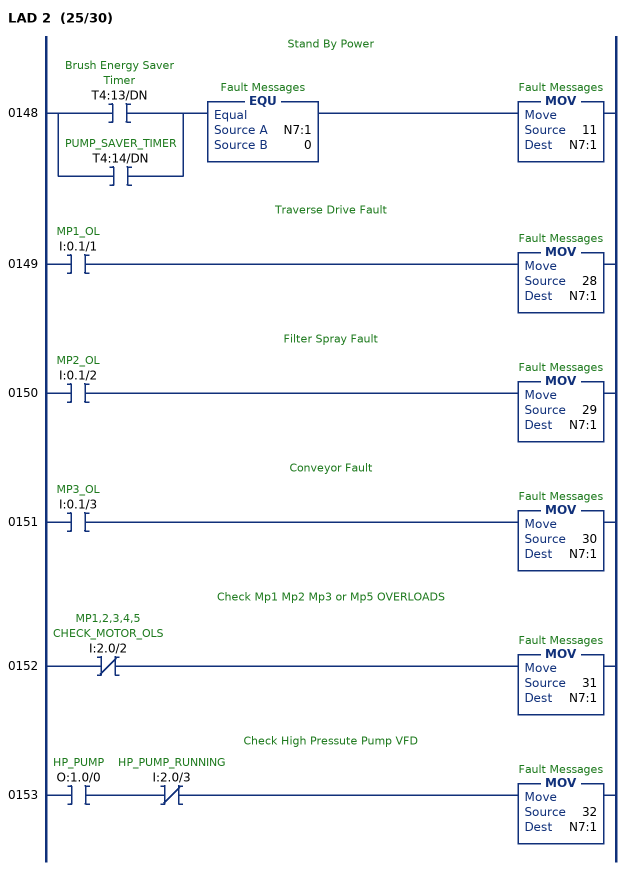
% Rung: 148 %
% Stand By Power %
SOR BST XIC T4:13/DN NXB XIC T4:14/DN BND EQU N7:1 0 MOV 11 N7:1 EOR
%   T4:13  "Brush Energy Saver Timer" %
%   T4:14/DN  PUMP_SAVER_TIMER %
%   N7:1  "Fault Messages" %
% Rung: 149 %
% Traverse Drive Fault %
SOR XIC I:0.1/1 MOV 28 N7:1 EOR
%   I:0.1/1  MP1_OL %
%   N7:1  "Fault Messages" %
% Rung: 150 %
% Filter Spray Fault %
SOR XIC I:0.1/2 MOV 29 N7:1 EOR
%   I:0.1/2  MP2_OL %
%   N7:1  "Fault Messages" %
% Rung: 151 %
% Conveyor Fault %
SOR XIC I:0.1/3 MOV 30 N7:1 EOR
%   I:0.1/3  MP3_OL %
%   N7:1  "Fault Messages" %
% Rung: 152 %
% Check Mp1 Mp2 Mp3 or Mp5 OVERLOADS %
SOR XIO I:2.0/2 MOV 31 N7:1 EOR
%   I:2.0/2  CHECK_MOTOR_OLS  "MP1,2,3,4,5" %
%   N7:1  "Fault Messages" %
% Rung: 153 %
% Check High Pressute Pump VFD %
SOR XIC O:1.0/0 XIO I:2.0/3 MOV 32 N7:1 EOR
%   O:1.0/0  HP_PUMP %
%   I:2.0/3  HP_PUMP_RUNNING %
%   N7:1  "Fault Messages" %

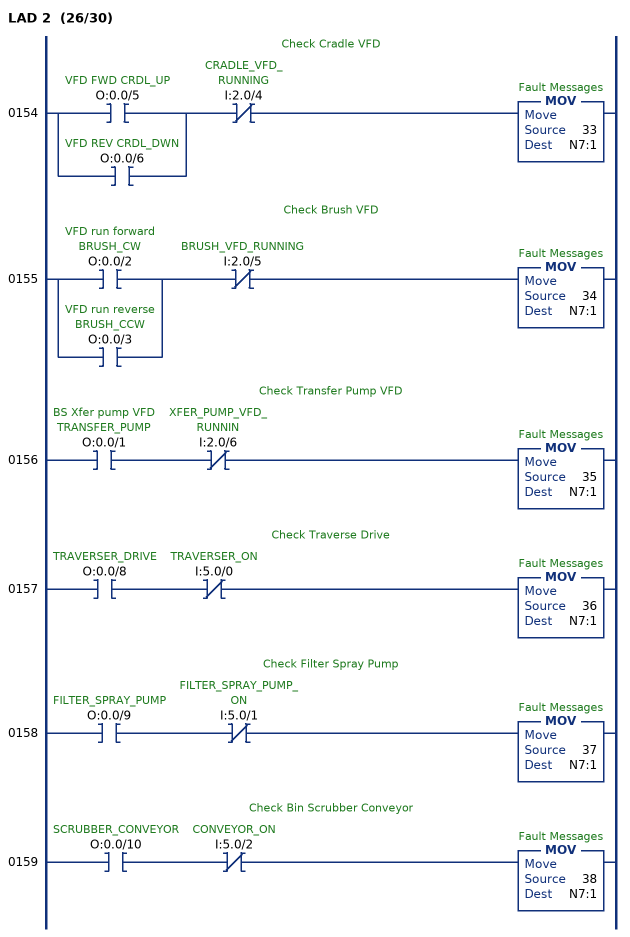
% Rung: 154 %
% Check Cradle VFD %
SOR BST XIC O:0.0/5 NXB XIC O:0.0/6 BND XIO I:2.0/4 MOV 33 N7:1 EOR
%   O:0.0/5  CRDL_UP  "VFD FWD" %
%   O:0.0/6  CRDL_DWN  "VFD REV" %
%   I:2.0/4  CRADLE_VFD_RUNNING %
%   N7:1  "Fault Messages" %
% Rung: 155 %
% Check Brush VFD %
SOR BST XIC O:0.0/2 NXB XIC O:0.0/3 BND XIO I:2.0/5 MOV 34 N7:1 EOR
%   O:0.0/2  BRUSH_CW  "VFD run forward" %
%   O:0.0/3  BRUSH_CCW  "VFD run reverse" %
%   I:2.0/5  BRUSH_VFD_RUNNING %
%   N7:1  "Fault Messages" %
% Rung: 156 %
% Check Transfer Pump VFD %
SOR XIC O:0.0/1 XIO I:2.0/6 MOV 35 N7:1 EOR
%   O:0.0/1  TRANSFER_PUMP  "BS Xfer pump VFD" %
%   I:2.0/6  XFER_PUMP_VFD_RUNNIN %
%   N7:1  "Fault Messages" %
% Rung: 157 %
% Check Traverse Drive %
SOR XIC O:0.0/8 XIO I:5.0/0 MOV 36 N7:1 EOR
%   O:0.0/8  TRAVERSER_DRIVE %
%   I:5.0/0  TRAVERSER_ON %
%   N7:1  "Fault Messages" %
% Rung: 158 %
% Check Filter Spray Pump %
SOR XIC O:0.0/9 XIO I:5.0/1 MOV 37 N7:1 EOR
%   O:0.0/9  FILTER_SPRAY_PUMP %
%   I:5.0/1  FILTER_SPRAY_PUMP_ON %
%   N7:1  "Fault Messages" %
% Rung: 159 %
% Check Bin Scrubber Conveyor %
SOR XIC O:0.0/10 XIO I:5.0/2 MOV 38 N7:1 EOR
%   O:0.0/10  SCRUBBER_CONVEYOR %
%   I:5.0/2  CONVEYOR_ON %
%   N7:1  "Fault Messages" %

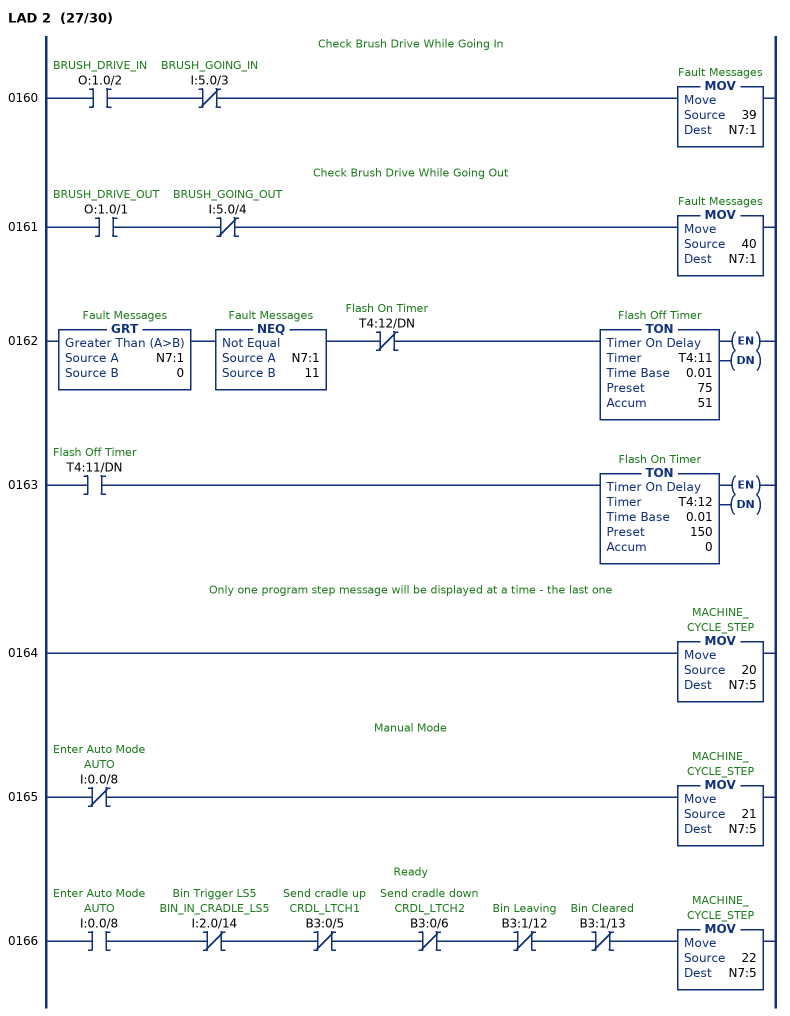
% Rung: 160 %
% Check Brush Drive While Going In %
SOR XIC O:1.0/2 XIO I:5.0/3 MOV 39 N7:1 EOR
%   O:1.0/2  BRUSH_DRIVE_IN %
%   I:5.0/3  BRUSH_GOING_IN %
%   N7:1  "Fault Messages" %
% Rung: 161 %
% Check Brush Drive While Going Out %
SOR XIC O:1.0/1 XIO I:5.0/4 MOV 40 N7:1 EOR
%   O:1.0/1  BRUSH_DRIVE_OUT %
%   I:5.0/4  BRUSH_GOING_OUT %
%   N7:1  "Fault Messages" %
% Rung: 162 %
SOR GRT N7:1 0 NEQ N7:1 11 XIO T4:12/DN TON T4:11 0.01 75 51 EOR
%   N7:1  "Fault Messages" %
%   T4:12  "Flash On Timer" %
%   T4:11  "Flash Off Timer" %
% Rung: 163 %
SOR XIC T4:11/DN TON T4:12 0.01 150 0 EOR
%   T4:11  "Flash Off Timer" %
%   T4:12  "Flash On Timer" %
% Rung: 164 %
% Only one program step message will be displayed at a time - the last one %
SOR MOV 20 N7:5 EOR
%   N7:5  MACHINE_CYCLE_STEP %
% Rung: 165 %
% Manual Mode %
SOR XIO I:0.0/8 MOV 21 N7:5 EOR
%   I:0.0/8  AUTO  "Enter Auto Mode" %
%   N7:5  MACHINE_CYCLE_STEP %
% Rung: 166 %
% Ready %
SOR XIC I:0.0/8 XIO I:2.0/14 XIO B3:0/5 XIO B3:0/6 XIO B3:1/12 XIO B3:1/13 MOV 22 N7:5 EOR
%   I:0.0/8  AUTO  "Enter Auto Mode" %
%   I:2.0/14  BIN_IN_CRADLE_LS5  "Bin Trigger LS5" %
%   B3:0/5  CRDL_LTCH1  "Send cradle up" %
%   B3:0/6  CRDL_LTCH2  "Send cradle down" %
%   B3:1/12  "Bin Leaving" %
%   B3:1/13  "Bin Cleared" %
%   N7:5  MACHINE_CYCLE_STEP %

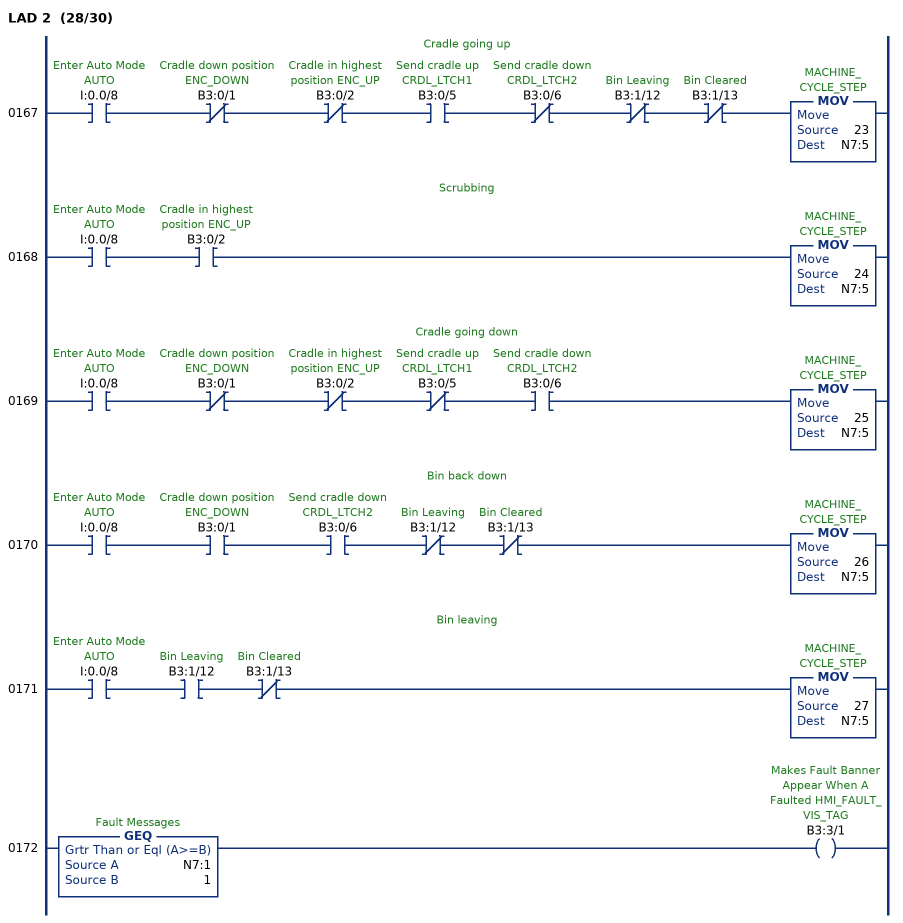
% Rung: 167 %
% Cradle going up %
SOR XIC I:0.0/8 XIO B3:0/1 XIO B3:0/2 XIC B3:0/5 XIO B3:0/6 XIO B3:1/12 XIO B3:1/13 MOV 23 N7:5 EOR
%   I:0.0/8  AUTO  "Enter Auto Mode" %
%   B3:0/1  ENC_DOWN  "Cradle down position" %
%   B3:0/2  ENC_UP  "Cradle in highest position" %
%   B3:0/5  CRDL_LTCH1  "Send cradle up" %
%   B3:0/6  CRDL_LTCH2  "Send cradle down" %
%   B3:1/12  "Bin Leaving" %
%   B3:1/13  "Bin Cleared" %
%   N7:5  MACHINE_CYCLE_STEP %
% Rung: 168 %
% Scrubbing %
SOR XIC I:0.0/8 XIC B3:0/2 MOV 24 N7:5 EOR
%   I:0.0/8  AUTO  "Enter Auto Mode" %
%   B3:0/2  ENC_UP  "Cradle in highest position" %
%   N7:5  MACHINE_CYCLE_STEP %
% Rung: 169 %
% Cradle going down %
SOR XIC I:0.0/8 XIO B3:0/1 XIO B3:0/2 XIO B3:0/5 XIC B3:0/6 MOV 25 N7:5 EOR
%   I:0.0/8  AUTO  "Enter Auto Mode" %
%   B3:0/1  ENC_DOWN  "Cradle down position" %
%   B3:0/2  ENC_UP  "Cradle in highest position" %
%   B3:0/5  CRDL_LTCH1  "Send cradle up" %
%   B3:0/6  CRDL_LTCH2  "Send cradle down" %
%   N7:5  MACHINE_CYCLE_STEP %
% Rung: 170 %
% Bin back down %
SOR XIC I:0.0/8 XIC B3:0/1 XIC B3:0/6 XIO B3:1/12 XIO B3:1/13 MOV 26 N7:5 EOR
%   I:0.0/8  AUTO  "Enter Auto Mode" %
%   B3:0/1  ENC_DOWN  "Cradle down position" %
%   B3:0/6  CRDL_LTCH2  "Send cradle down" %
%   B3:1/12  "Bin Leaving" %
%   B3:1/13  "Bin Cleared" %
%   N7:5  MACHINE_CYCLE_STEP %
% Rung: 171 %
% Bin leaving %
SOR XIC I:0.0/8 XIC B3:1/12 XIO B3:1/13 MOV 27 N7:5 EOR
%   I:0.0/8  AUTO  "Enter Auto Mode" %
%   B3:1/12  "Bin Leaving" %
%   B3:1/13  "Bin Cleared" %
%   N7:5  MACHINE_CYCLE_STEP %
% Rung: 172 %
SOR GEQ N7:1 1 OTE B3:3/1 EOR
%   N7:1  "Fault Messages" %
%   B3:3/1  HMI_FAULT_VIS_TAG  "Makes Fault Banner Appear When A Faulted" %

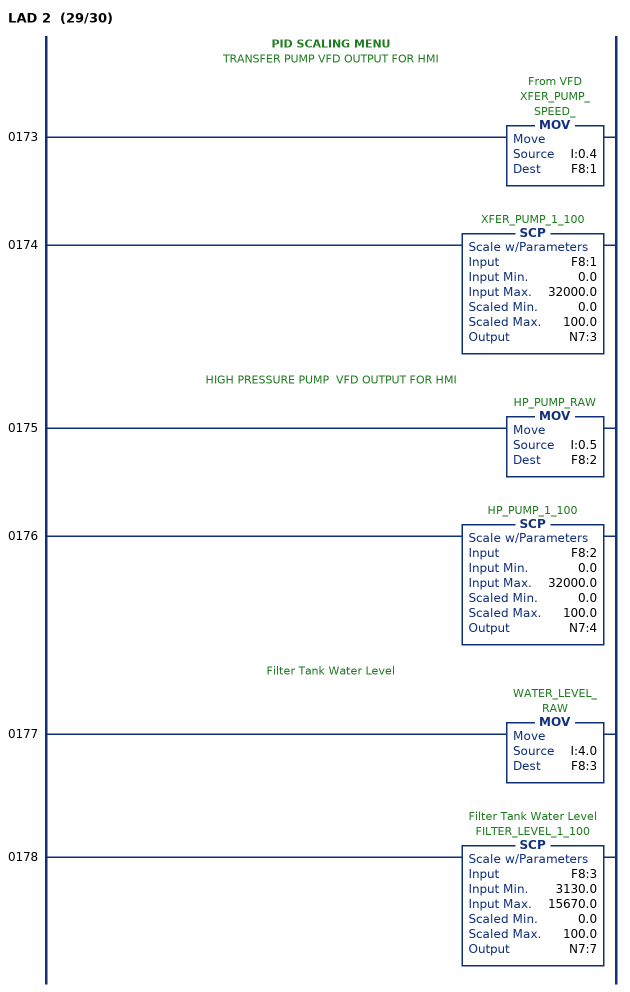
% Rung: 173 %
% TITLE: PID SCALING MENU %
% TRANSFER PUMP VFD OUTPUT FOR HMI %
SOR MOV I:0.4 F8:1 EOR
%   I:0.4  TRANSFER_PUMP_SPEED  "0/10v" %
%   F8:1  XFER_PUMP_SPEED_  "From VFD" %
% Rung: 174 %
SOR SCP F8:1 0.0 32000.0 0.0 100.0 N7:3 EOR
%   F8:1  XFER_PUMP_SPEED_  "From VFD" %
%   N7:3  XFER_PUMP_1_100 %
% Rung: 175 %
% HIGH PRESSURE PUMP  VFD OUTPUT FOR HMI %
SOR MOV I:0.5 F8:2 EOR
%   I:0.5  HP_PUMP_SPEED  "0/10v" %
%   F8:2  HP_PUMP_RAW %
% Rung: 176 %
SOR SCP F8:2 0.0 32000.0 0.0 100.0 N7:4 EOR
%   F8:2  HP_PUMP_RAW %
%   N7:4  HP_PUMP_1_100 %
% Rung: 177 %
% Filter Tank Water Level %
SOR MOV I:4.0 F8:3 EOR
%   I:4.0  XFER_TANK_LEVEL  "Raw Value" %
%   F8:3  WATER_LEVEL_RAW %
% Rung: 178 %
SOR SCP F8:3 3130.0 15670.0 0.0 100.0 N7:7 EOR
%   F8:3  WATER_LEVEL_RAW %
%   N7:7  FILTER_LEVEL_1_100  "Filter Tank Water Level" %

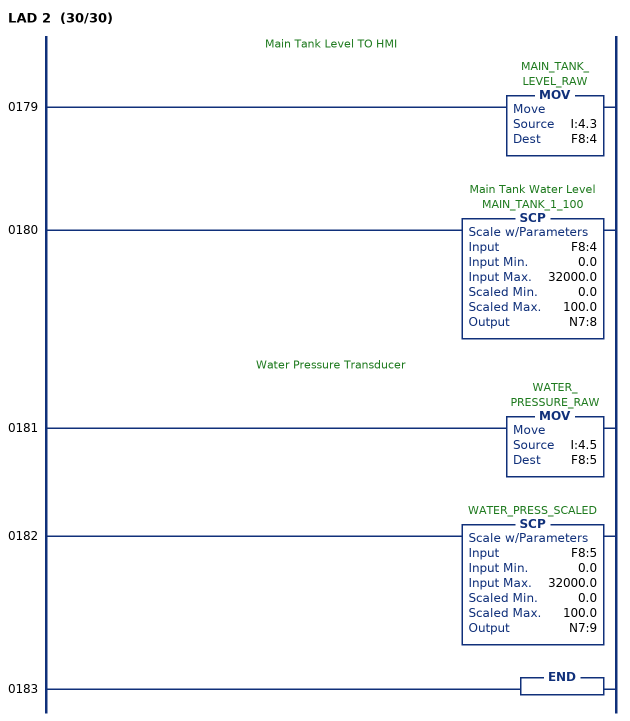
% Rung: 179 %
% Main Tank Level TO HMI %
SOR MOV I:4.3 F8:4 EOR
%   I:4.3  WATER_PRESSURE_SENS  "Pressure Sensor" %
%   F8:4  MAIN_TANK_LEVEL_RAW %
% Rung: 180 %
SOR SCP F8:4 0.0 32000.0 0.0 100.0 N7:8 EOR
%   F8:4  MAIN_TANK_LEVEL_RAW %
%   N7:8  MAIN_TANK_1_100  "Main Tank Water Level" %
% Rung: 181 %
% Water Pressure Transducer %
SOR MOV I:4.5 F8:5 EOR
%   F8:5  WATER_PRESSURE_RAW %
% Rung: 182 %
SOR SCP F8:5 0.0 32000.0 0.0 100.0 N7:9 EOR
%   F8:5  WATER_PRESSURE_RAW %
%   N7:9  WATER_PRESS_SCALED %
% Rung: 183 %
SOR END EOR

OTHER DOCUMENTED ADDRESSES
  B3:4/2  MANIFOLD_ONS
  B3:4/3  MANIFOLD_DELAY_ONS
  B3:4/4  MANIFOLD_ONS_
  B3:4/5  MANIFOLD_DELAY_ONS_
  F8:7  PRESSURE_SENS_RAW
  N7:12  RAW_XFER_TANK_LEVEL
  N7:13  KC_
  N7:14  TI
  N7:15  TD
  N7:16  LUT
  N7:17  HMI_WATER_LEVEL_SP  "0-100"
  N7:18  PID_SET_POINT  "WATER LEVEL 0-16383"
  N7:19  PID_PV_WATER_LEVEL  "RAW WATER LEVEL TO PID SCALED VALUE"
  N7:21  PID_OUTPUT_RAW  "0-16383"
  N7:22  PID_OUTPUT_FOR_VFD  "0-32000"
  N7:23  HMI_MANUAL_RUN
  N7:24  HP_PUMP_SP  "HMI SP"
  N7:25  HP_KC_SP
  N7:26  HP_TI_SP
  N7:27  HP_TD_SP
  N7:28  HP_LUT_SP
  N7:29  HMI_PRESSURE_SP  "HP PUMP PRESSURE SP"
  N7:30  HP_PUMP_SP_PID  "HMI SETPOINT FOR PID"
  N7:31  PRESSURE_FOR_PID_PV
  N7:33  HP_PID_OUTPUT_  "TO HP VFD 0-32000"
  N7:34  HMI_MANUAL_HP_SPEED  "HMI MANUAL RUN SPEED FOR HP PUMP"
  N7:35  HMI_ACTUAL_PRESSURE
  N7:39  HP_SPEED_CRADLE_UP
  N7:40  BIN_SIZING_HMI  "INFORMS HMI BIN SIZE"
  O:0.0  XFER_PUMP_VFD_OUTPUT
  O:0.1  OUT_TO_HP_VFD
  O:3.0/1  PALLET_WASH_DOWN  "Pallet Manifold Down SOL"
  O:3.0/3  BIN_26_CLAMP_ON  "Cradle Clamp"
  PD11:0  PID_FOR_XFER_PUMP  "BIN SCRUBBER TRANSFER PUMP"
  PD11:1.2  PRESSURE_SP
  PD11:1.3  HP_KC
  PD11:1.4  HP_TI
  PD11:1.5  HP_TD
  PD11:1.13  LOOP_UPDATE_TIME  ".002"
  T4:25  MANIFOLD_DELAY_TMR  "Slows HP Pump for a few seconds"

DATA TABLE (non-zero values as saved)
DATA B3
% B3:0 % 0X010B 0X0800 0X0730 0X0002 0XBD00 0X0000
DATA T4
% .PRE .ACC %
% T4:0 % 50 50
% T4:3 % 500 0
% T4:4 % 2 2
% T4:9 % 2 2
% T4:11 % 75 51
% T4:12 % 150 0
% T4:13 % 120 52
% T4:14 % 120 52
% T4:15 % 5 0
% T4:16 % 5 0
% T4:17 % 500 0
% T4:18 % 2 2
% T4:25 % 4 4
% T4:26 % 50 50
% T4:27 % 15 15
DATA N7
% N7:0 % 0 38 0 0 0 22 27 77 0 0
% N7:10 % 0 0 12739 50 1 0 2 0 0 12604
% N7:20 % 77 0 0 0 0 0 0 0 0 0
% N7:30 % 0 -8175 0 0 0 -175 0 0 0 0
% N7:40 % 4
DATA F8
% F8:0 % 0 0 0 12739 4
% F8:5 % 0 0 4
